Staubli VAL3: orderDistance.pgx

program orderDistance(num& x_nValue[] (dimensions=1), num x_nCoeff (dimensions=1))
  local num l_nValue[4]
  local num i
begin
  //
  // x_nValue[0]= home index
  // x_nValue[1]= joint index
  // x_nValue[2]= nDistance
  // x_nCoeff = coefficent using J4 J5 J6
  //
  // INIT
  //
  // copy
  l_nValue=x_nValue
  l_nValue[1]=x_nValue[1]
  l_nValue[2]=x_nValue[2]
  l_nValue[3]=x_nCoeff
  //
  if nDistance==-1
    nDistance=x_nValue[2]
    nJoint=x_nValue[1]
    nHome=x_nValue
    nCoeff=x_nCoeff
  else
    // MAKE THE  LIST
    for i=0 to size(nDistance)-1
      // a minimum find
      if x_nValue[2]<nDistance[i]
        call insertValue(l_nValue,i)
        return
      else
        // not found put at the end
        if i==size(nDistance)-1
          call insertValue(l_nValue,i+1)
          return
        endIf
      endIf
    endFor
  endIf
end
